// TIA Portal V20 export
DATA_BLOCK "GLOBAL_PP_HMI_IF_DB"   // DB210
{ S7_Optimized_Access := 'TRUE' }
// stored: AutoNumber false, MemoryReserve 100
   VAR
      PP : Array[0..50] of "TEC_UNIT_HMI_UDT";
      Hide_PP_Check : Array[0..50] of Bool;
      Check_TON : Array[0..50] of TON_TIME;
   END_VAR
BEGIN
   // PP[0] : 放卷上位
   // PP[1] : +ST020-CNV06-VM01-PX01 / 放卷下位
   // PP[2] : +ST020-CNV06-VM01-PX02 / +ST010-TL02- PP01
   // PP[3] : +ST020-CNV06-VM01-PX03 / +ST010-TL02- PP02
   // PP[4] : +ST020-TL01- PP01
   // PP[5] : +ST020-CNV06-VM01-PX05 / +ST020-TL01- PP02
   // PP[6] : +ST020-CNV06-VM01-PX06 / +ST020-TL02- PP01
   // PP[7] : +ST020-CNV06-VM01-PX07 / +ST020-TL02- PP02
   // PP[8] : +ST020-CNV06-VM01-PX08
   // PP[9] : +ST020-CNV06-VM01-PX09
   // PP[10] : +ST020-CNV06-VM01-PX10
   // PP[11] : +ST020-CNV06-VM01-PX11
   // PP[12] : +ST020-CNV06-VM01-PX20
   // PP[13] : +ST020-CNV06-VM01-PEY01
   // PP[14] : +ST020-CNV06-VM01-PEY02
   // PP[15] : +ST020-CNV06-VM01-PEY03
   // PP[16] : +ST020-CNV06-VM01-PEY04
   // PP[17] : +ST020-CNV06-PX21
   // PP[18] : +ST020-CNV06-PX12
   // PP[20] : +ST020-CNV04-VM01-PX01 Unload Pos1
   // PP[21] : +ST020-CNV04-VM01-PX02 Unload Pos2
   // PP[22] : +ST020-CNV04-VM01-PX03 Unload Pos3
   // PP[23] : +ST020-CNV04-VM01-PX04 WaitPos1 Off
   // PP[24] : +ST020-CNV04-VM01-PX05 WaitPos1
   // PP[25] : +ST020-CNV04-VM01-PX06 WaitPos2 Off
   // PP[26] : +ST020-CNV04-VM01-PX07 WaitPos2
   // PP[27] : +ST020-CNV04-VM01-PX08 WaitPos2 Full
   // PP[28] : +ST020-CNV04-VM01-PX09 WaitPos3 Off
   // PP[29] : +ST020-CNV04-VM01-PX10 WaitPos3
   // PP[30] : +ST020-CNV04-VM01-PX11 WaitPos3 Full
   // PP[31] : +ST020-CNV04-VM01-PX12 WaitPos4 Off
   // PP[32] : +ST020-CNV04-VM01-PX13 WaitPos4
   // PP[33] : +ST020-CNV04-VM01-PX17 LoadPos Off
   // PP[34] : +ST020-CNV04-VM01-PX14 LoadPos1
   // PP[35] : +ST020-CNV04-VM01-PX15 LoadPos2
   // PP[36] : +ST020-CNV04-VM01-PX16 LoadPos3
   // PP[37] : +ST020-CNV04-VM01-PX19 LoadPos4
   // PP[38] : +ST020-CNV04-VM01-PX18 LoadposBypass
   // PP[39] : +ST020-CNV04-VM01-PX20 LoadPos Ready
   // PP[40] : +ST020-CNV04-VM01-PX21 Unload Pos
   // PP[41] : +ST020-CNV04-VM01-PX36 Chain Check
   // PP[42] : +ST020-CNV04-VM01-PX37 Load Slide Table Check
   // PP[43] : +ST020-CNV04-VM01-PX38 Unload Slide Table Check
   // PP[44] : +ST020-CNV04-VM01-PEY01 Unload Part Check
   // PP[45] : +ST020-CNV04-VM01-PEY02 Unload Part Check
   // PP[46] : +ST020-CNV04-VM01-PEY03 Load Part Check
   // PP[47] : +ST020-CNV04-VM01-PEY04 Load Part Check
   // PP[48] : +ST020-CNV04-VM01-PX22 Unload Pos Full
   // PP[50] : +ST020-TL12-SX02
   // Hide_PP_Check[1] : +ST020-CNV06-VM01-PX01
   // Hide_PP_Check[2] : +ST020-CNV06-VM01-PX02
   // Hide_PP_Check[3] : +ST020-CNV06-VM01-PX03
   // Hide_PP_Check[5] : +ST020-CNV06-VM01-PX05
   // Hide_PP_Check[6] : +ST020-CNV06-VM01-PX06
   // Hide_PP_Check[7] : +ST020-CNV06-VM01-PX07
   // Hide_PP_Check[8] : +ST020-CNV06-VM01-PX08
   // Hide_PP_Check[9] : +ST020-CNV06-VM01-PX09
   // Hide_PP_Check[10] : +ST020-CNV06-VM01-PX10
   // Hide_PP_Check[11] : +ST020-CNV06-VM01-PX11
   // Hide_PP_Check[12] : +ST020-CNV06-VM01-PX20
   // Hide_PP_Check[13] : +ST020-CNV06-VM01-PEY01
   // Hide_PP_Check[14] : +ST020-CNV06-VM01-PEY02
   // Hide_PP_Check[15] : +ST020-CNV06-VM01-PEY03
   // Hide_PP_Check[16] : +ST020-CNV06-VM01-PEY04
   // Hide_PP_Check[17] : +ST020-CNV06-PX21
   // Hide_PP_Check[20] : +ST020-CNV04-VM01-PX01 Unload Pos1
   // Hide_PP_Check[21] : +ST020-CNV04-VM01-PX02 Unload Pos2
   // Hide_PP_Check[22] : +ST020-CNV04-VM01-PX03 Unload Pos3
   // Hide_PP_Check[23] : +ST020-CNV04-VM01-PX04 WaitPos1 Off
   // Hide_PP_Check[24] : +ST020-CNV04-VM01-PX05 WaitPos1
   // Hide_PP_Check[25] : +ST020-CNV04-VM01-PX06 WaitPos2 Off
   // Hide_PP_Check[26] : +ST020-CNV04-VM01-PX07 WaitPos2
   // Hide_PP_Check[27] : +ST020-CNV04-VM01-PX08 WaitPos2 Full
   // Hide_PP_Check[28] : +ST020-CNV04-VM01-PX09 WaitPos3 Off
   // Hide_PP_Check[29] : +ST020-CNV04-VM01-PX10 WaitPos3
   // Hide_PP_Check[30] : +ST020-CNV04-VM01-PX11 WaitPos3 Full
   // Hide_PP_Check[31] : +ST020-CNV04-VM01-PX12 WaitPos4 Off
   // Hide_PP_Check[32] : +ST020-CNV04-VM01-PX13 WaitPos4
   // Hide_PP_Check[33] : +ST020-CNV04-VM01-PX17 LoadPos Off
   // Hide_PP_Check[34] : +ST020-CNV04-VM01-PX14 LoadPos1
   // Hide_PP_Check[35] : +ST020-CNV04-VM01-PX15 LoadPos2
   // Hide_PP_Check[36] : +ST020-CNV04-VM01-PX16 LoadPos3
   // Hide_PP_Check[37] : +ST020-CNV04-VM01-PX19 LoadPos4
   // Hide_PP_Check[38] : +ST020-CNV04-VM01-PX18 LoadposBypass
   // Hide_PP_Check[39] : +ST020-CNV04-VM01-PX20 LoadPos Ready
   // Hide_PP_Check[40] : +ST020-CNV04-VM01-PX21 Unload Pos
   // Hide_PP_Check[41] : +ST020-CNV04-VM01-PX36 Chain Check
   // Hide_PP_Check[42] : +ST020-CNV04-VM01-PX37 Load Slide Table Check
   // Hide_PP_Check[43] : +ST020-CNV04-VM01-PX38 Unload Slide Table Check
   // Hide_PP_Check[44] : +ST020-CNV04-VM01-PEY01 Unload Part Check
   // Hide_PP_Check[45] : +ST020-CNV04-VM01-PEY02 Unload Part Check
   // Hide_PP_Check[46] : +ST020-CNV04-VM01-PEY03 Load Part Check
   // Hide_PP_Check[47] : +ST020-CNV04-VM01-PEY04 Load Part Check
   // Hide_PP_Check[48] : +ST020-CNV04-VM01-PX22 Unload Pos Full
   // Hide_PP_Check[50] : +ST020-TL12-SX02
   // Check_TON[1] : +ST020-CNV06-VM01-PX01
   // Check_TON[2] : +ST020-CNV06-VM01-PX02
   // Check_TON[3] : +ST020-CNV06-VM01-PX03
   // Check_TON[5] : +ST020-CNV06-VM01-PX05
   // Check_TON[6] : +ST020-CNV06-VM01-PX06
   // Check_TON[7] : +ST020-CNV06-VM01-PX07
   // Check_TON[8] : +ST020-CNV06-VM01-PX08
   // Check_TON[9] : +ST020-CNV06-VM01-PX09
   // Check_TON[10] : +ST020-CNV06-VM01-PX10
   // Check_TON[11] : +ST020-CNV06-VM01-PX11
   // Check_TON[12] : +ST020-CNV06-VM01-PX20
   // Check_TON[13] : +ST020-CNV06-VM01-PEY01
   // Check_TON[14] : +ST020-CNV06-VM01-PEY02
   // Check_TON[15] : +ST020-CNV06-VM01-PEY03
   // Check_TON[16] : +ST020-CNV06-VM01-PEY04
   // Check_TON[17] : +ST020-CNV06-PX21
   // Check_TON[20] : +ST020-CNV04-VM01-PX01 Unload Pos1
   // Check_TON[21] : +ST020-CNV04-VM01-PX02 Unload Pos2
   // Check_TON[22] : +ST020-CNV04-VM01-PX03 Unload Pos3
   // Check_TON[23] : +ST020-CNV04-VM01-PX04 WaitPos1 Off
   // Check_TON[24] : +ST020-CNV04-VM01-PX05 WaitPos1
   // Check_TON[25] : +ST020-CNV04-VM01-PX06 WaitPos2 Off
   // Check_TON[26] : +ST020-CNV04-VM01-PX07 WaitPos2
   // Check_TON[27] : +ST020-CNV04-VM01-PX08 WaitPos2 Full
   // Check_TON[28] : +ST020-CNV04-VM01-PX09 WaitPos3 Off
   // Check_TON[29] : +ST020-CNV04-VM01-PX10 WaitPos3
   // Check_TON[30] : +ST020-CNV04-VM01-PX11 WaitPos3 Full
   // Check_TON[31] : +ST020-CNV04-VM01-PX12 WaitPos4 Off
   // Check_TON[32] : +ST020-CNV04-VM01-PX13 WaitPos4
   // Check_TON[33] : +ST020-CNV04-VM01-PX17 LoadPos Off
   // Check_TON[34] : +ST020-CNV04-VM01-PX14 LoadPos1
   // Check_TON[35] : +ST020-CNV04-VM01-PX15 LoadPos2
   // Check_TON[36] : +ST020-CNV04-VM01-PX16 LoadPos3
   // Check_TON[37] : +ST020-CNV04-VM01-PX19 LoadPos4
   // Check_TON[38] : +ST020-CNV04-VM01-PX18 LoadposBypass
   // Check_TON[39] : +ST020-CNV04-VM01-PX20 LoadPos Ready
   // Check_TON[40] : +ST020-CNV04-VM01-PX21 Unload Pos
   // Check_TON[41] : +ST020-CNV04-VM01-PX36 Chain Check
   // Check_TON[42] : +ST020-CNV04-VM01-PX37 Load Slide Table Check
   // Check_TON[43] : +ST020-CNV04-VM01-PX38 Unload Slide Table Check
   // Check_TON[44] : +ST020-CNV04-VM01-PEY01 Unload Part Check
   // Check_TON[45] : +ST020-CNV04-VM01-PEY02 Unload Part Check
   // Check_TON[46] : +ST020-CNV04-VM01-PEY03 Load Part Check
   // Check_TON[47] : +ST020-CNV04-VM01-PEY04 Load Part Check
   // Check_TON[48] : +ST020-CNV04-VM01-PX22 Unload Pos Full
   // Check_TON[50] : +ST020-TL12-SX02
END_DATA_BLOCK
